// SIMATIC S7-200 SMART project (STEP 7-Micro/WIN SMART), CPU SR40

ORGANIZATION_BLOCK 主程序:OB1
TITLE=程序注释
BEGIN
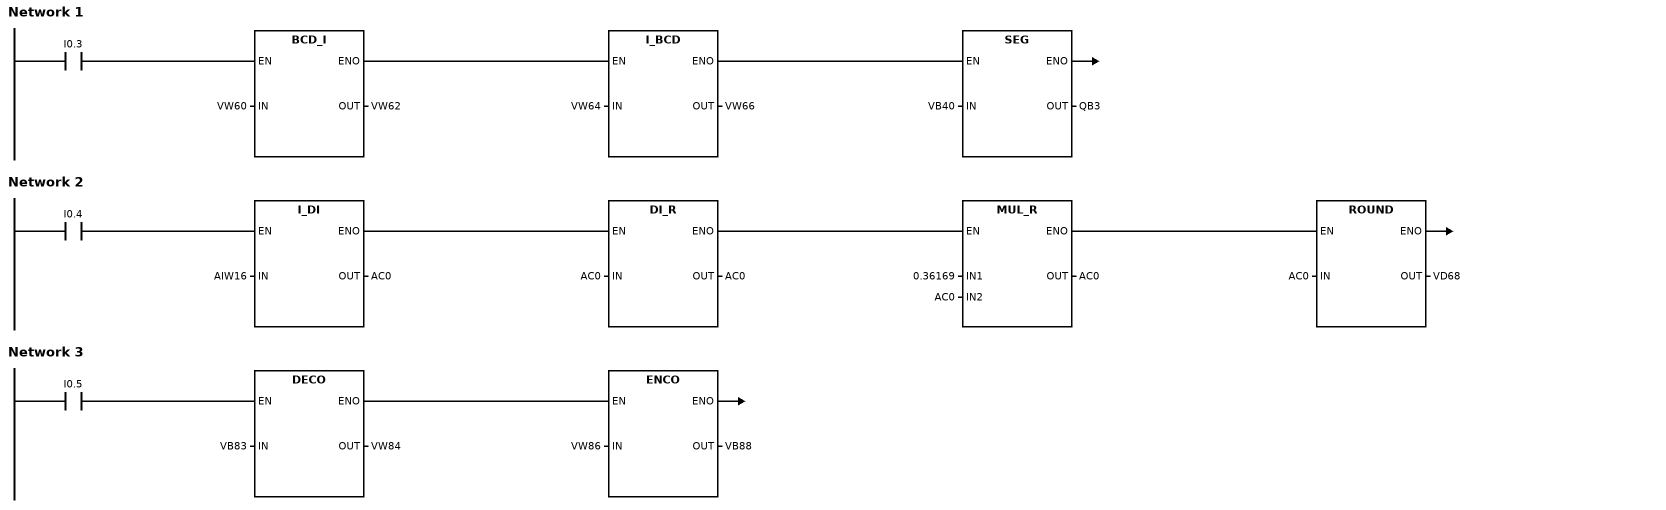
Network 1
LD     I0.3
MOVW   VW60, VW62
AENO
BCDI   VW62
AENO
MOVW   VW64, VW66
AENO
IBCD   VW66
AENO
SEG    VB40, QB3
Network 2
LD     I0.4
ITD    AIW16, AC0
AENO
DTR    AC0, AC0
AENO
*R     0.36169, AC0
AENO
ROUND  AC0, VD68
Network 3
LD     I0.5
DECO   VB83, VW84
AENO
ENCO   VW86, VB88
END_ORGANIZATION_BLOCK
